Staubli VAL3: loadCycle.pgx

public program loadCycle(string x_sItem, num& x_nResult[])
  local string l_sName
  local string l_sPath
  local string l_sType
begin
  call getType(l_sType)
  // load it
  if find(saveProg:libPath(),saveData:sPathProg)==-1
    x_nResult=saveProg:libLoad(saveData:sPathProg+l_sType)
    delay(0)
    if saveData:bDebug
      ? "loading PROG..."+saveData:sPathProg+l_sType
    endIf
    // check if exist or not
  endIf
  // reload the edit template
  if isDefined(saveProg:pProg[x_sItem].sID) and x_sItem!=""
    // refresh the iD...
    saveProg:pProg[x_sItem].sID=x_sItem
    // item found
    x_nResult=0
  endIf
end
